// TIA Portal V16 program export: 1 tag tables, 0 data types, 0 data blocks, 2 code blocks (in call order from the OBs), 0 instance data blocks

VAR_GLOBAL   // PLC tag table "Tabla de variables estándar"
END_VAR

ORGANIZATION_BLOCK "Main"   // OB1, LAD, ProgramCycle
TITLE = "Main Program Sweep (Cycle)"
{ S7_Optimized_Access := 'TRUE' }
VERSION : 0.1
// stored: AutoNumber true, IsIECCheckEnabled false, SetENOAutomatically false
   VAR_INPUT
      Initial_Call : Bool;   // Initial call of this OB
      Remanence : Bool;   // =True, if remanent data are available
   END_VAR
BEGIN
END_ORGANIZATION_BLOCK

FUNCTION "DBReset" : Void
{ S7_Optimized_Access := 'TRUE' }
VERSION : 0.1
   VAR_INPUT 
      dbNumber : DInt;
      Nvariables : Int;
   END_VAR

   VAR_IN_OUT 
      sdfsd : Bool;
      sdfsdf : Bool;
      sdfsdf_1 : Bool;
      sdfsdf_2 : Bool;
      sdfsdf_3 : Bool;
      sdfsdf_4 : Bool;
   END_VAR

   VAR_TEMP 
      "db" : DB_ANY;
      _byteOffset : Int;
      _bitOffset : Int;
   END_VAR


BEGIN
	//Si Nvariables = 0. Reset de totes les variables del db a l'array.
	//Si Nvariables <>0. Es fa Reset del número de LWORDS des del començament del DB fins a l'Array.
	
	#db := UINT_TO_DB_ANY(WORD_TO_UINT(DINT_TO_WORD(#dbNumber)));
	
	IF #Nvariables = 0 THEN
	    
	    FOR #_byteOffset := 0 TO ("ALARMES_SIZE_ARRAY" * 8) DO
	        FOR #_bitOffset := 0 TO 7 DO
	            POKE_BOOL(area := 16#84,
	                      dbNumber := 250,
	                      byteOffset := #_byteOffset,
	                      bitOffset := #_bitOffset,
	                      value := FALSE,
	                      ENO => ENO);
	        END_FOR;
	    END_FOR;
	    
	ELSE
	    
	    FOR #_byteOffset := 0 TO (#Nvariables * 8) DO
	        FOR #_bitOffset := 0 TO 7 DO
	            POKE_BOOL(area := 16#84,
	                      dbNumber := 250,
	                      byteOffset := #_byteOffset,
	                      bitOffset := #_bitOffset,
	                      value := FALSE,
	                      ENO => ENO);
	        END_FOR;
	    END_FOR;
	    
	END_IF;
	
	
	
END_FUNCTION
